FUNCTION_BLOCK HW_Control_Core (* Basic FB with empty ECC *)
  (* Standard: 61499-2 *)
  (* Version 1.0, 2023-03-02, AK125171 *)
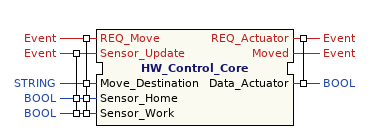
  EVENT_INPUT
    REQ_Move WITH Move_Destination, Sensor_Home, Sensor_Work;
    Sensor_Update WITH Sensor_Home, Sensor_Work;
  END_EVENT
  EVENT_OUTPUT
    REQ_Actuator WITH Data_Actuator;
    Moved;
  END_EVENT
  VAR_INPUT
    Move_Destination : STRING;
    Sensor_Home : BOOL;
    Sensor_Work : BOOL;
  END_VAR
  VAR_OUTPUT
    Data_Actuator : BOOL;
  END_VAR
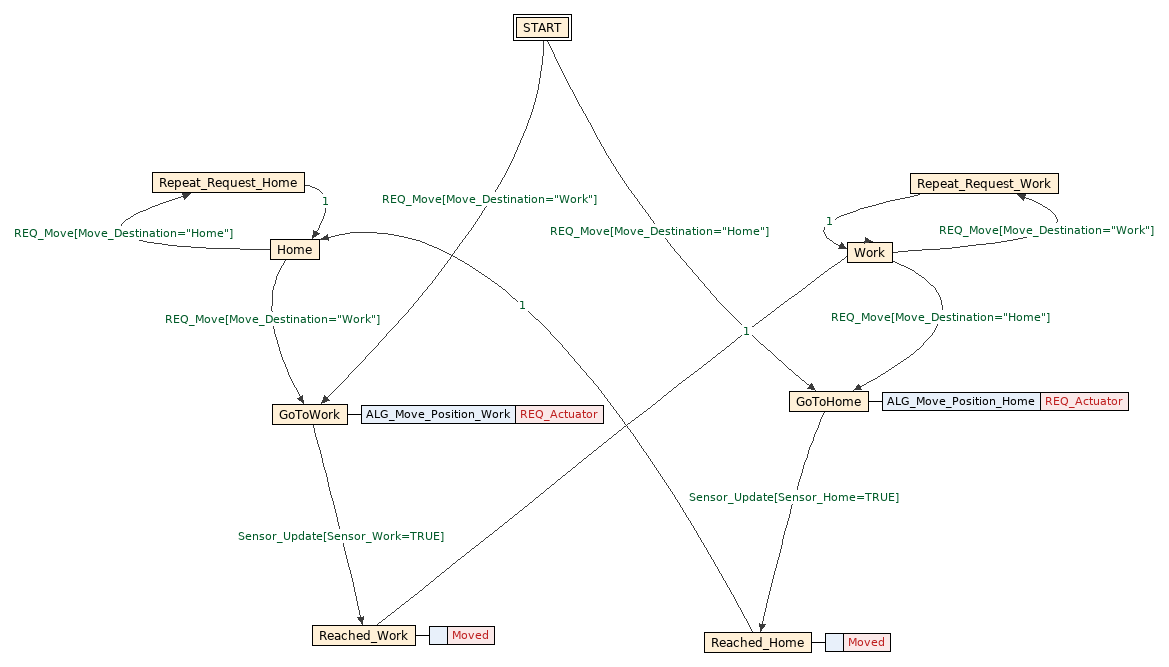
  EC_STATES
    START; (* Initial State *)
    GoToHome : ALG_Move_Position_Home -> REQ_Actuator;
    GoToWork : ALG_Move_Position_Work -> REQ_Actuator;
    Home;
    Work;
    Reached_Work : -> Moved;
    Reached_Home : -> Moved;
    Repeat_Request_Home;
    Repeat_Request_Work;
  END_STATES
  EC_TRANSITIONS
    Home TO GoToWork := REQ_Move[Move_Destination="Work"];
    Work TO GoToHome := REQ_Move[Move_Destination="Home"];
    GoToWork TO Reached_Work := Sensor_Update[Sensor_Work=TRUE];
    GoToHome TO Reached_Home := Sensor_Update[Sensor_Home=TRUE];
    Reached_Work TO Work := 1;
    Reached_Home TO Home := 1;
    Home TO Repeat_Request_Home := REQ_Move[Move_Destination="Home"];
    Work TO Repeat_Request_Work := REQ_Move[Move_Destination="Work"];
    Repeat_Request_Home TO Home := 1;
    Repeat_Request_Work TO Work := 1;
    START TO GoToWork := REQ_Move[Move_Destination="Work"];
    START TO GoToHome := REQ_Move[Move_Destination="Home"];
  END_TRANSITIONS
  ALGORITHM ALG_Move_Position_Home IN ST: (* Sets Data_Move FALSE for Event REQ_Move "Home" *)
Data_Actuator:=FALSE;
  END_ALGORITHM
  ALGORITHM ALG_Move_Position_Work IN ST: (* Sets Data_Move TRUE for Event REQ_Move "Work" *)
Data_Actuator:=TRUE;
  END_ALGORITHM
END_FUNCTION_BLOCK
